Staubli VAL3: getNextID.pgx

public program getNextID(num x_nConvNum (dimensions=1), num& x_nNextID[] (dimensions=1))
begin
  // This program returns the number of the next available ID
  //
  // Input Param
  //  x_nConvNum  : Conveyor number
  //
  // Output Param
  //  x_nNextID : value of the next partID in the stack
  //        -1 --> No Part Available
  //
  //----------------------------------------------------------------
  //
  switch x_nConvNum
    case 0
      call cnv0:getNextID(x_nNextID)
    break
    case 1
      call cnv1:getNextID(x_nNextID)
    break
  endSwitch
end
